// TIA Portal V15.1 export
// export: Created 2026-01-15T16:29:38.1606694Z, ExportSetting WithDefaults, WithReadOnly, DisplayName Totally Integrated Automation Portal, DisplayVersion V15.1 Update 8, DisplayName TIA Portal Openness, DisplayVersion V15.1 Update 8, DisplayName STEP 7 Professional, DisplayVersion V15.1 Update 8, DisplayName WinCC Advanced, DisplayVersion V15.1 Update 8
FUNCTION "1. CONVER TC" : Void   // FC1, LAD
{ S7_Optimized_Access := 'TRUE' }
VERSION : 0.1
// stored: AutoNumber true, CodeModifiedDate 2025-08-27T17:05:49.4204143Z, CompileDate 2026-01-15T16:25:52.7071747Z, CreationDate 2026-01-15T16:22:49.8270549Z, HandleErrorsWithinBlock false, InterfaceModifiedDate 2024-10-18T04:03:55.072308Z, IsConsistent true, IsIECCheckEnabled false, IsKnowHowProtected false, IsWriteProtected false, LibraryConformanceStatus The object is library-conformant., ModifiedDate 2025-08-27T17:05:49.4204143Z, ParameterModified 2024-10-18T04:03:55.072308Z, PLCSimAdvancedSupport false, SetENOAutomatically False, StructureModified 2024-10-18T04:03:55.072308Z, UDAEnableTagReadback false
   VAR_INPUT
      AI : Int;
      HS : Real;
   END_VAR
   VAR_OUTPUT
      TEMP_OUT : Real;
      XUNG_OUT : Real;
   END_VAR
   VAR_TEMP
      AI_REAL : Real;
   END_VAR
BEGIN

REGION Network 1
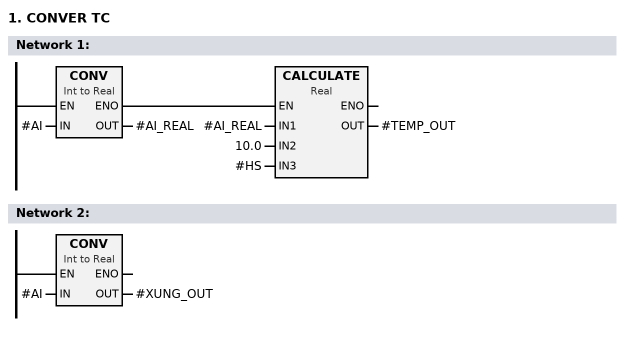
   RUNG wire#powerrail
      { S7_Templates := "[SrcType := Int, DestType := Real]" } Convert(in := #AI, out => #AI_REAL)
      { S7_Templates := "SrcType := Real"; S7_Expression := "(IN1/IN2)*IN3" } Calculate(in1 := #AI_REAL, in2 := 10.0, in3 := #HS, out => #TEMP_OUT)
   END_RUNG
   // the same network as SCL:
   #AI_REAL := INT_TO_REAL(#AI);
   #TEMP_OUT := (#AI_REAL/10.0)*#HS;
END_REGION

REGION Network 2
   RUNG wire#powerrail
      { S7_Templates := "[SrcType := Int, DestType := Real]" } Convert(in := #AI, out => #XUNG_OUT)
   END_RUNG
   // the same network as SCL:
   #XUNG_OUT := INT_TO_REAL(#AI);
END_REGION
END_FUNCTION
